TYPE Lens_Struct :
STRUCT
	IN :    BOOL;
	KNOWN : BOOL;
END_STRUCT
END_TYPE

(* stored: Version 1.1.0.1, ProductVersion 3.1.4018.5
   DUT Lens_Struct: Id {36c64e89-932e-4d90-91ea-396f68cbc675} *)
